FUNCTION strcpy : UDINT
VAR_INPUT
	pDst : POINTER TO STRING;
	pSrc : POINTER TO STRING;
END_VAR
VAR
	pArr		: POINTER TO BYTE;
	pArrDst		: POINTER TO BYTE;
END_VAR

pArr		:= pSrc;
pArrDst		:= pDst;
WHILE (pArr^ <> 0)  DO
	pArrDst^ := pArr^;

	pArr := pArr+1;
	pArrDst := pArrDst+1;

END_WHILE
pArrDst^ := pArr^;

END_FUNCTION

(* stored: Version 1.1.0.1, ProductVersion 3.1.4024.3
   POU strcpy: Id {97a10faa-b44c-0dc2-0a81-046bed0613f2}, SpecialFunc None *)
